# EPICS substitutions: template/mtcaevr300_ess.substitutions
#
# Micro-Research Finland Oy mTCA.4 Event Receiver
# This is the standard ESS EVR for MTCA crate : mTCA-EVR-300
#
#
# nat> show_fruinfo 7
# ---------------------------------------
# FRU Info for device 7:
# ---------------------------------------
# Common Header    : 0x01 0x00 0x00 0x01 0x0c 0x19 0x00 0xd9
# ---------------------------------------
# Internal Use Area : -
# ---------------------------------------
# Chassis Info Area : -
# ---------------------------------------
# Board Info Area          : at offs=8, len=88
# Manufacturer(25)         : Micro-Research Finland Oy
# Board Name(12)           : mTCA-EVR-300
# Serial Number(07)        : P376053
# Part Number(12)          : mTCA-EVR-300
# FRU file ID(16)          : mtcaevr300dc.fru
# ---------------------------------------
# Product Info Area        : at offs=96, len=104
# Manufacturer(25)         : Micro-Research Finland Oy
# Product Name(21)         : mTCA.4 Event Receiver
# Product Number(12)       : mTCA-EVR-300
# Part Version(04)         : v1.1
# Product Serial Number(07): P376053
# Asset Tag(00)            :  -
# FRU file ID(16)          : mtcaevr300dc.fru
# ---------------------------------------
#
# nat> show_sensorinfo 7
# Sensor Information for FRU 7 / AMC3
# ==================================================================
#   #   SDRType  Sensor Entity Inst  Value   State    Name
# ------------------------------------------------------------------
#   -   MDevLoc          0xc1  0x63                    mTCA-EVR-300
#   0   Full     0xf2    0xc1  0x63  0x04              Hot Swap
#   1   Full     Voltage 0xc1  0x63  2.368 V    ok     REF
#   2   Full     Voltage 0xc1  0x63  5.9 V      ok     Temp 1
#   3   Full     Voltage 0xc1  0x63  0.5 V      ok     Temp 2
#   4   Full     Voltage 0xc1  0x63  0.992 V    ok     1.0 V
#   5   Full     Voltage 0xc1  0x63  1.776 V    ok     1.8 V
#   6   Full     Voltage 0xc1  0x63  12.3 V     ok     12 V
#   7   Full     Voltage 0xc1  0x63  3.296 V    ok     3.3 V
#   8   Full     Voltage 0xc1  0x63  3.200 V    ok     3.3 V MP
#   9   Compact  0x0b    0xc1  0x63  0x00              0x00  FPGA Done
#  10   Full     Temp    0xc1  0x63  28.0 C     ok     Local
#  11   Full     Temp    0xc1  0x63  39.0 C     ok     FPGA
#  12   Compact  0xf0    0xc1  0x63  0x10              HS 007 AMC3
# --------------------

global {dev=$(_PREF), link=$(_SESS), id=$(_ID), fruid=$(_FRUID)}

file "fru_common_ess.template"
{
pattern { unit          }
        { $(_UNIT)      }
}

file "sensor_ai_ess.template"
{
pattern { attr,         sensinst,   type,   prefix          }
        { RefV,         1,          2,      $(_ID)$(_UNIT)  }
        { Temp1V,       2,          2,      $(_ID)$(_UNIT)  }
        { Temp2V,       3,          2,      $(_ID)$(_UNIT)  }
        { 1d0V,         4,          2,      $(_ID)$(_UNIT)  }
        { 1d8V,         5,          2,      $(_ID)$(_UNIT)  }
        { 12dV,         6,          2,      $(_ID)$(_UNIT)  }
        { 3d3V,         7,          2,      $(_ID)$(_UNIT)  }
        { Mp3d3V,       8,          2,      $(_ID)$(_UNIT)  }
        { LocalTemp,    1,          1,      $(_ID)$(_UNIT)  }
        { FpgaTemp,     2,          1,      $(_ID)$(_UNIT)  }
}
